// TIA Portal V20 export
VAR_GLOBAL   // PLC tag table "LGR_Const_Task_CommandType"
END_VAR
VAR_GLOBAL CONSTANT   // user constants
   CMD_POWER_ON : Byte := 16#20;
   CMD_DRIVE_ON : Byte := 16#21;
   CMD_CHANGE_SPEED : Byte := 16#2A;
   CMD_TASK_UP : Byte := 16#40;
   CMD_TASK_PICK : Byte := 16#41;
   CMD_TASK_DROP : Byte := 16#42;
   CMD_TASK_MOVE : Byte := 16#43;
   CMD_TASK_MEASURE : Byte := 16#44;   // Measure task (MeasureItem / MeasureSku / MeasureFloor flags). Move = avoidance move only, R10 / 측정 작업 (MeasureItem / MeasureSku / MeasureFloor 플래그로 세부 지정). Move 는 회피 이동 전용, R10
   CMD_TASK_AVOID_REF : Byte := 16#4A;
   CMD_TASK_AVOID_ABS : Byte := 16#4B;
   CMD_TASK_AVOID_REL : Byte := 16#4C;
   CMD_TASK_RESERVED_0x4D : Byte := 16#4D;
   CMD_TASK_MODIFY : Byte := 16#4E;
   CMD_TASK_DELETE : Byte := 16#4F;
   CMD_STOP_FAST : Byte := 16#50;
   CMD_STOP_NORMAL : Byte := 16#51;
   CMD_STOP_CYCLE : Byte := 16#52;
   CMD_RESERVED_0x53 : Byte := 16#53;
   CMD_INITIALIZING : Byte := 16#54;
   CMD_HOMING : Byte := 16#55;
   CMD_MOVE_TO_ORIGIN_CELL : Byte := 16#56;
   CMD_MOVE_TO_MAINT_POSITION : Byte := 16#57;
   CMD_CHANGE_MODE : Byte := 16#60;
   CMD_CHANGE_PARA_GANTRY : Byte := 16#70;
   CMD_CHANGE_PARA_COMPONENT : Byte := 16#71;
   CMD_REQUEST_STATUS_GANTRY : Byte := 16#30;
   CMD_DRIVE_JOG : Byte := 16#25;
   CMD_TEACHING : Byte := 16#80;
   CMD_TEACHING_ITEM : Byte := 16#82;
END_VAR
